PROGRAM MAIN
VAR
END_VAR

ModbusRTU();
MQTT();

END_PROGRAM

(* stored: Version 1.1.0.1, ProductVersion 3.1.4024.12
   POU MAIN: Id {cbe6a41c-6ffc-4215-aca8-6d4f58f1cfe4}, SpecialFunc None *)
